(* IEC 61131-3 sources: library-inventory-agv/src/global_variables, 2 files *)

(* ---- GVL_Main.st ---- *)
// =============================================================================
// GVL_Main — Core Application Variables
// =============================================================================

{attribute 'qualified_only'}
VAR_GLOBAL
    // =========================================================================
    // AGV Master Control
    // =========================================================================
    fbAgvControl    : AgvControl_FB;        // Master state machine instance
    eAgvState       : E_AgvState;           // Current AGV state (mirrored for HMI)

    // =========================================================================
    // Navigation Waypoints
    // =========================================================================
    aPointsName     : ARRAY[0..99] OF STRING(80);   // Navigation point names
    aPointsName01   : ARRAY[0..99] OF STRING(80);   // Alternate point list
    aPointChargingName : STRING(80) := 'Charging_01'; // Charging station point
    aPointHomeName     : STRING(80) := 'Home_01';     // Home/standby point
    spointsName     : STRING(80);           // Currently active point name
    iPointCount     : INT;                  // Total waypoints in current task
    nPointPosition  : INT;                  // Current waypoint index

    // =========================================================================
    // Task Management
    // =========================================================================
    sTask_Number    : STRING(40);           // Current task ID
    sTask_Number1   : STRING(40);           // Previous task ID
    nAreaCount      : INT;                  // Number of areas to scan
    nCurrentArea    : INT;                  // Current area index

    // =========================================================================
    // Shelf Configuration (loaded from HMI_BookShelfSeting)
    // =========================================================================
    stCurrentShelf  : ST_ShelfConfig;       // Active shelf parameters

    // =========================================================================
    // Sensor Clients
    // =========================================================================
    fbRfidClient    : SensorTcpClient;      // RFID reader TCP connection
    fbVisionClient  : SensorTcpClient;      // Vision camera TCP connection

    // =========================================================================
    // Communication Status
    // =========================================================================
    bNavSystemOnline    : BOOL;             // Navigation API reachable
    bNodeRedOnline      : BOOL;             // Node-RED data store reachable
    bRfidConnected      : BOOL;             // RFID reader TCP connected
    bVisionConnected    : BOOL;             // Vision camera TCP connected
    bRobConnected       : BOOL;             // Scanning mechanism connected

    // =========================================================================
    // Modbus I/O Mirrors
    // =========================================================================
    bEStopActive    : BOOL;                 // Emergency stop pressed
    bAx01_PowerOn   : BOOL;                 // Axis 01 enable output
    bAx02_PowerOn   : BOOL;                 // Axis 02 enable output
    bLight01_On     : BOOL;                 // Warning light 1
    bLight02_On     : BOOL;                 // Warning light 2

    // =========================================================================
    // Diagnostics
    // =========================================================================
    udiMainTaskCycCount : UDINT;            // Cycle counter (overflow = ~49 days at 10ms)
    tSystemUptime       : TIME;             // System uptime
END_VAR

(* ---- GVL_Servo.st ---- *)
// =============================================================================
// GVL_Servo — Servo/Stepper Axis Configuration and Runtime Parameters
// =============================================================================

{attribute 'qualified_only'}
VAR_GLOBAL
    // =========================================================================
    // Axis References
    // =========================================================================
    // Physical EtherCAT axes connected to XINJE DP3C(L) drives.
    // AXIS_REF_ETC_DS402_CS provides the SoftMotion interface for
    // Cyclic Synchronous Position mode over EtherCAT.

    stAxis01        : AXIS_REF_ETC_DS402_CS;    // Vertical lift axis
    stAxis02        : AXIS_REF_ETC_DS402_CS;    // Secondary axis

    // =========================================================================
    // Dynamic Limits — Applied to all motion commands
    // =========================================================================

    // Velocity limits (mm/s)
    fMaxVelocity    : LREAL := 500.0;       // Maximum travel speed
    fMaxVelKeep     : LREAL := 300.0;       // Cruising speed during steady travel
    fMaxVelTurn     : LREAL := 100.0;       // Speed limit during direction reversal

    // Acceleration limits (mm/s²)
    fMaxAcceleration : LREAL := 800.0;      // Maximum acceleration
    fMaxDeceleration : LREAL := 800.0;      // Maximum deceleration

    // Jerk limit (mm/s³) — controls S-curve smoothness
    // Higher jerk = faster transition but more vibration
    // Lower jerk  = smoother but slower acceleration ramp
    fMaxJerk        : LREAL := 3000.0;

    // =========================================================================
    // Protection Limits
    // =========================================================================

    // Following error threshold (mm)
    // If |commanded_pos - actual_pos| exceeds this value, axis enters ErrorStop.
    // This detects: mechanical obstruction, belt slip, encoder fault, motor stall.
    fMaxPositionLag : LREAL := 5.0;

    // Force limits (drive-specific)
    fMaxTorque      : LREAL := 3.0;         // Nm (stepper rated torque)
    fMaxCurrent     : LREAL := 5.0;         // Amps (drive current limit)

    // =========================================================================
    // Preset Positions (mm)
    // =========================================================================
    // Quick-access positions for HMI jog/preset buttons.

    rAx01_PresetP01 : LREAL := 0.0;        // Bottom position (home)
    rAx01_PresetP02 : LREAL := 1800.0;     // Top position (full travel)
    rAx02_PresetP01 : LREAL := 0.0;
    rAx02_PresetP02 : LREAL := 1800.0;

    // =========================================================================
    // Jog Velocities (mm/s) — Operator-adjustable from HMI
    // =========================================================================
    fAx01_JogVel    : LREAL := 50.0;       // Default jog speed axis 1
    fAx02_JogVel    : LREAL := 50.0;       // Default jog speed axis 2

    // =========================================================================
    // Runtime Status (read-only from application code)
    // =========================================================================
    bAx01_Enabled   : BOOL;                // Axis 1 powered
    bAx01_Homed     : BOOL;                // Axis 1 homing complete
    bAx01_Moving    : BOOL;                // Axis 1 in motion
    bAx01_Error     : BOOL;                // Axis 1 fault active
    rAx01_ActPos    : LREAL;               // Axis 1 actual position (mm)
    rAx01_ActVel    : LREAL;               // Axis 1 actual velocity (mm/s)

    bAx02_Enabled   : BOOL;
    bAx02_Homed     : BOOL;
    bAx02_Moving    : BOOL;
    bAx02_Error     : BOOL;
    rAx02_ActPos    : LREAL;
    rAx02_ActVel    : LREAL;
END_VAR
